TYPE (* Encapsulated interlock interface: Count + the InterlockRule array *)
  (* Standard: 1131-3 *)
  (* Version 0.1, 6/21/2026, easensoy, WMG, single STRUCT input wrapping the rule count and rules *)
  PACKAGE Main;
  InterlockTable : STRUCT
    Count : INT;
    Rules : ARRAY [{{RuleArraySize}}] OF InterlockRule;
  END_STRUCT;
END_TYPE
